INTERFACE I_ExtensionAddedEvent EXTENDS I_Event

PROPERTY PUBLIC Target : I_Extension
GET
END_GET
END_PROPERTY

END_INTERFACE

(* stored: Version 1.1.0.1, ProductVersion 3.1.4024.12
   Itf I_ExtensionAddedEvent: Id {dbd2a8df-e169-4e6c-b3fb-4a98208ff3ca}
   Property Target: Id {c9d623ce-ed79-4a58-8e3b-d8a0bb20ce33}
   Get Get: Id {7ed110af-ffef-42ca-9b7c-abb4e8070b7b} *)
